(*********************************** G.D S.p.A. - Technical Department ***********************************
============= PROGRAM INFO ============
FOLDER:             TBD
MACHINES INVOLVED:  TBD 

============= DESCRIPTION =============
Low task

============= REVISIONS ===============
Date		Version	 	Author      	Description             
----------	-------		------------  	--------------------------------------------
2019/03/28 	0000.00	 	CEC 			Creation of the PRG

**********************************************************************************************************)

PROGRAM _csp_customerInterfaces_highest
VAR
END_VAR

;

END_PROGRAM

(* stored: Version 1.1.0.1, ProductVersion 3.1.4022.12
   POU _csp_customerInterfaces_highest: Id {6da1d8b5-a758-49b5-9eeb-730a35212709}, SpecialFunc None *)
